FUNCTION F_CheckPistonPosition : E_ErrorModes
VAR_INPUT
END_VAR
VAR
END_VAR

// Check if piston is out of bounds
IF HMI.fCylinderPositonReference > Parameters.stPistonRange.fPistonPosMax THEN
	HMI.fCylinderPositonReference := Parameters.stPistonRange.fPistonPosMax;	
	HMI.sPistonEndStopMessage := Parameters.stPistonOutOfBounds.sPistonMax;
	Parameters.eErrorModes := E_ErrorModes.MaxLimit;
	HMI.sPistonEndStopMessage := Parameters.stPistonOutOfBounds.sPistonMax;
	Parameters.stStateVariables.fTime := 0.0;
ELSIF HMI.fCylinderPositonReference < Parameters.stPistonRange.fPistonPosMin  THEN
	HMI.fCylinderPositonReference := Parameters.stPistonRange.fPistonPosMin;
	Parameters.eErrorModes := E_ErrorModes.MinLimit;
	HMI.sPistonEndStopMessage := Parameters.stPistonOutOfBounds.sPistonMin;
	Parameters.stStateVariables.fTime := 0.0;
ELSE
	HMI.sPistonEndStopMessage := Parameters.stPistonOutOfBounds.sNotActive;
	Parameters.eErrorModes := E_ErrorModes.NaN;
END_IF

END_FUNCTION

(* stored: Version 1.1.0.1, ProductVersion 3.1.4024.10
   POU F_CheckPistonPosition: Id {6f408e8f-58a0-4a52-a52a-6c9eb15374a1}, SpecialFunc None *)
